# EPICS substitutions: evrSupport/Db/ioc/IOC-LI21-RF01bsa.substitutions
# BSA records
#
# One per device:
# Please check the HOPR,LOPR,PREC,ADEL,MDEL values provided in bsaPHASEdef.db!
file bsaPHASEdef.db {
#      Device               ,loc'n , IOC  , system, Attribute
  pattern {DEVICE           , LOC  ,  UN  , SYS   , ATRB   , EF    }
	  { ACCL:LI21:1         , LI21 , RF01 , SYS0  , L1S_P  , _L1S_P}
	  { ACCL:LI21:180       , LI21 , RF01 , SYS0  , L1X_P  , _L1X_P}
	  { PCAV:LI21:300       , LI21 , RF01 , SYS0  , P      , _P    }
}
# One per device:
# Please check the HOPR,LOPR,PREC,ADEL,MDEL values provided in bsaAMPLEdef.db!
file bsaAMPLEdef.db {
#      Device               ,loc'n , IOC  ,system , Attribute
  pattern {DEVICE           , LOC  ,  UN  , SYS   , ATRB  ,  EF   }
	  { ACCL:LI21:1         , LI21 , RF01 , SYS0  , L1S_A , _L1S_A}
	  { ACCL:LI21:180       , LI21 , RF01 , SYS0  , L1X_A , _L1X_A}
	  { PCAV:LI21:300       , LI21 , RF01 , SYS0  , A     , _A    }
